{attribute 'qualified_only'}
{attribute 'to_string'}
TYPE Chipboard :
(
	CIP18 := 1,
	CIP54,
	
	size
);
END_TYPE

(* stored: Version 1.1.0.1, ProductVersion 3.1.4024.11
   DUT Chipboard: Id {3cb4f29c-803e-4d95-bc5f-59e240b5a1eb} *)
